Staubli VAL3: observeStop.pgx

program observeStop()
begin
  //**************************************************
  // Method interrupts a running move operation. This is
  // equivalent to a pause.
  //
  // Method is triggered by a flag being set.
  // N.B. Move is only stopped until flag is unset.
  //**************************************************
  while true
    wait(moveIsStopped==true)
    stopMove()
    wait(moveIsStopped==false)
    restartMove()
  endWhile
end
